{attribute 'GeneratedUsingTerminal: EK1100-0000-0018'}
{attribute addProperty BoxType "EK1100-0000-0018"}
{attribute addProperty Id "Beckhoff_APS4xxxEK1122Beckhoff_APS4xxxEK1122_9CDB7635276A_0002_APS4322_5000_0017APS4322_A49C5437320"}
{attribute addProperty CRC "1989420928"}
{attribute addProperty Size "596"}
TYPE Beckhoff_APS4xxx_76942780 EXTENDS EK1100_1FC0878B :
STRUCT
	{attribute addProperty Name "Beckhoff_APS4xxxEK1122"}
	{attribute addProperty PreviousPort "Beckhoff APS4xxx : B"}
	Beckhoff_APS4xxxEK1122 : Beckhoff_APS4xxxEK1122_9CDB7635;
	{attribute addProperty Name "A_0002_APS4322_5000_0017"}
	{attribute addProperty PreviousPort "Beckhoff APS4xxxEK1122 : C"}
	A_0002_APS4322_5000_0017 : APS4322_A49C5437;
END_STRUCT
END_TYPE

(* stored: Version 1.2.0.0, ProductVersion 3.1.4024.9
   DUT Beckhoff_APS4xxx_76942780: Id {7c7a31ab-72d6-4367-a20d-6d5eb4c2e66d} *)
